{attribute 'no_explicit_call' := 'do not call this POU directly'} 
FUNCTION_BLOCK DigitalInput_NO
VAR
	DI_Input						AT %I*: BOOL;
END_VAR

PROPERTY isOff : bool
GET
isOff 		:= NOT DI_Input;
END_GET
END_PROPERTY

PROPERTY isOn : bool
GET
isOn			:= DI_Input;
END_GET
END_PROPERTY

END_FUNCTION_BLOCK

(* stored: Version 1.1.0.1
   POU DigitalInput_NO: Id {0b2b6594-9ed1-49ff-a036-d754db32d580}, SpecialFunc None
   Property isOff: Id {6ab52287-2ac7-4c78-818f-b6c32152155f}
   Get Get: Id {94a52a54-7745-47c6-8232-b056cd9b5e19}
   Property isOn: Id {e47d8458-2000-4994-917c-85221325622d}
   Get Get: Id {8819dc3c-76fb-49e8-ace3-ec88a172e7ba} *)
